(* Schneider Machine Expert - Basic project atividade2, file version 2.7.0.0 *)
(* ProjectInformations: Name=Novo projeto *)

HARDWARE
  Cpu 0: TM221CE24R
  EthernetConfiguration: NetworkName=M221, IpAllocationMode=FixedAddress, IpAddress=0.0.0.0, SubnetMask=0.0.0.0
  SerialLineConfiguration: Baud=Baud19200, Parity=ParityEven, DataBits=DataBits8, StopBits=StopBits1, PhysicalMedium=PhysicalMediumRs485, TransmissionMode=TransmissionModeModbusRtu, SlaveId=1, Addressing=SlaveAddressing
  MastTask: UsePeriodScanMode=false, PeriodScan=100
  FastTask: Period=255
  CpuBehavior: StartingMode=StartAsPreviousState, AutoSaveRamOnEeprom=true, WatchdogPeriod=250

SYMBOLS  (address, symbol, comment, settings)
  %M0       SIG_IN_SEN_A_ATU
  %M1       SIG_IN_SEN_A_DESA
  %M2       SIG_IN_SEN_B_ATU
  %M3       SIG_IN_SEN_B_DESA
  %M4       SIG_IN_SEN_C_ATU
  %M5       SIG_IN_SEN_C_DESA
  %M6       SIG_IN_SEN_D_ATU
  %M7       SIG_IN_SEN_D_DESA
  %M10      SIG_OUT_M1_LIGA
  %M11      SIG_OUT_M1_DESL
  %M12      SIG_OUT_M2_LIGA
  %M13      SIG_OUT_M2_DESL
  %M14      SIG_OUT_P1_LIGA
  %M15      SIG_OUT_P1_DESL
  %M16      SIG_OUT_AL1_LIGA
  %M17      SIG_OUT_AL1_DESL
  %M20      SIG_OUT_M1
  %M21      SIG_OUT_M2
  %M22      SIG_OUT_P1
  %M23      SIG_OUT_P2
  %M24      SIG_OUT_SEN_A
  %M25      SIG_OUT_SEN_B
  %M26      SIG_OUT_SEN_C
  %M27      SIG_OUT_SEN_D
  %M30      SIN_IN_SEL_A_ATU
  %M31      SIN_IN_SEL_A_DESA
  %M32      SIN_IN_EMERG_ATU
  %M33      SIN_IN_EMERG_DESA
  %I0.0     IN_SEN_A
  %I0.1     IN_SEN_B
  %I0.2     IN_SEN_C
  %I0.3     IN_SEN_D
  %I0.4     IN_SEL_A_ATU
  %I0.5     IN_SEL_A_DESA
  %I0.6     IN_EMERG_ATU
  %I0.7     IN_EMERG_DESA
  %Q0.0     OUT_M1
  %Q0.1     OUT_M2
  %Q0.2     OUT_P1
  %Q0.3     OUT_AL1
  %Q0.4     OUT_SEN_A
  %Q0.5     OUT_SEN_B
  %Q0.6     OUT_SEN_C
  %Q0.7     OUT_SEN_D

POU Entradas
  (* SectionNumber=1 *)

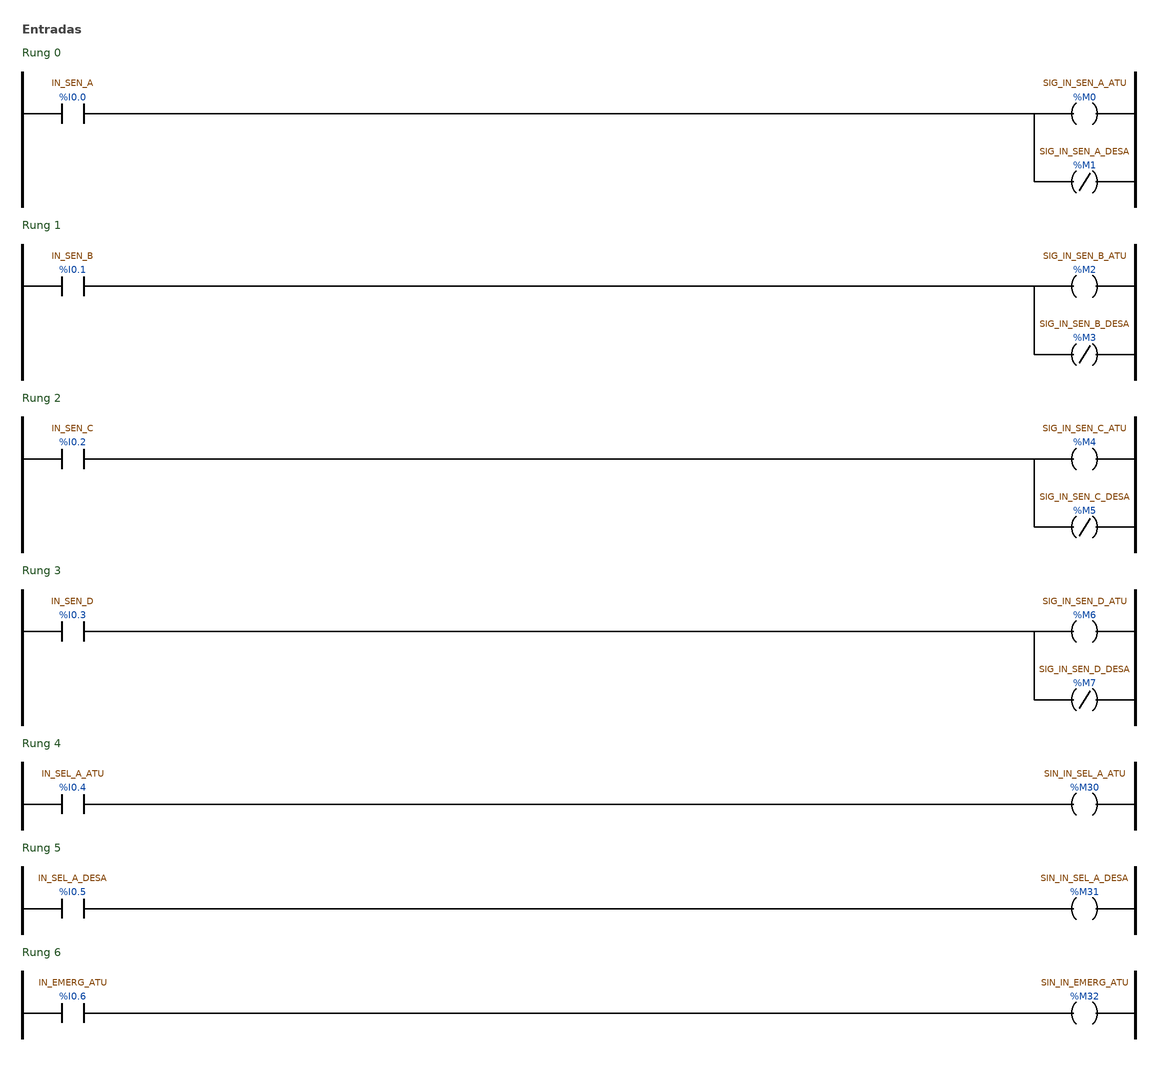

// Rung 0
  LD %I0.0                (* IN_SEN_A *)
  ST %M0                  (* SIG_IN_SEN_A_ATU *)
  STN %M1                 (* SIG_IN_SEN_A_DESA *)
  // as ST:
  //   SIG_IN_SEN_A_ATU := IN_SEN_A;
  //   SIG_IN_SEN_A_DESA := NOT IN_SEN_A;

// Rung 1
  LD %I0.1                (* IN_SEN_B *)
  ST %M2                  (* SIG_IN_SEN_B_ATU *)
  STN %M3                 (* SIG_IN_SEN_B_DESA *)
  // as ST:
  //   SIG_IN_SEN_B_ATU := IN_SEN_B;
  //   SIG_IN_SEN_B_DESA := NOT IN_SEN_B;

// Rung 2
  LD %I0.2                (* IN_SEN_C *)
  ST %M4                  (* SIG_IN_SEN_C_ATU *)
  STN %M5                 (* SIG_IN_SEN_C_DESA *)
  // as ST:
  //   SIG_IN_SEN_C_ATU := IN_SEN_C;
  //   SIG_IN_SEN_C_DESA := NOT IN_SEN_C;

// Rung 3
  LD %I0.3                (* IN_SEN_D *)
  ST %M6                  (* SIG_IN_SEN_D_ATU *)
  STN %M7                 (* SIG_IN_SEN_D_DESA *)
  // as ST:
  //   SIG_IN_SEN_D_ATU := IN_SEN_D;
  //   SIG_IN_SEN_D_DESA := NOT IN_SEN_D;

// Rung 4
  LD %I0.4                (* IN_SEL_A_ATU *)
  ST %M30                 (* SIN_IN_SEL_A_ATU *)
  // as ST:
  //   SIN_IN_SEL_A_ATU := IN_SEL_A_ATU;

// Rung 5
  LD %I0.5                (* IN_SEL_A_DESA *)
  ST %M31                 (* SIN_IN_SEL_A_DESA *)
  // as ST:
  //   SIN_IN_SEL_A_DESA := IN_SEL_A_DESA;

// Rung 6
  LD %I0.6                (* IN_EMERG_ATU *)
  ST %M32                 (* SIN_IN_EMERG_ATU *)
  // as ST:
  //   SIN_IN_EMERG_ATU := IN_EMERG_ATU;

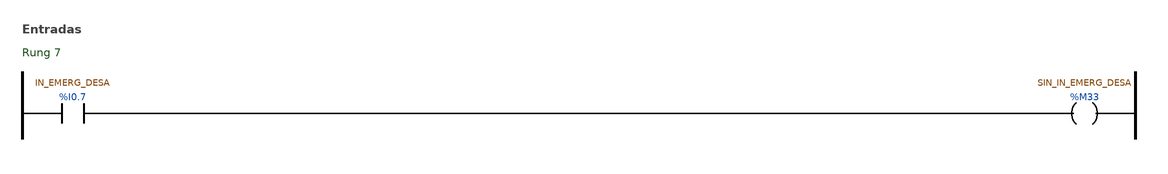

// Rung 7
  LD %I0.7                (* IN_EMERG_DESA *)
  ST %M33                 (* SIN_IN_EMERG_DESA *)
  // as ST:
  //   SIN_IN_EMERG_DESA := IN_EMERG_DESA;

POU Lógica
  (* SectionNumber=2 *)

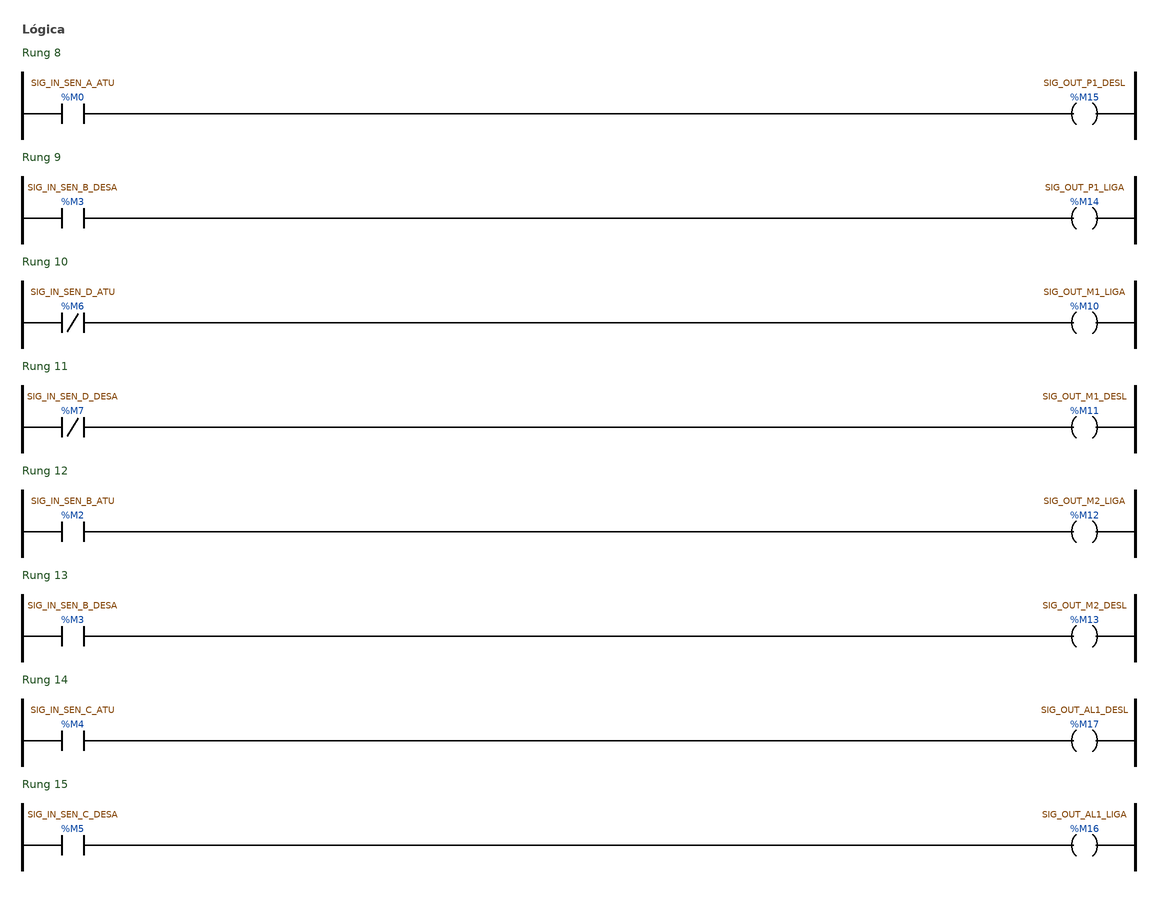

// Rung 8
  LD %M0                  (* SIG_IN_SEN_A_ATU *)
  ST %M15                 (* SIG_OUT_P1_DESL *)
  // as ST:
  //   SIG_OUT_P1_DESL := SIG_IN_SEN_A_ATU;

// Rung 9
  LD %M3                  (* SIG_IN_SEN_B_DESA *)
  ST %M14                 (* SIG_OUT_P1_LIGA *)
  // as ST:
  //   SIG_OUT_P1_LIGA := SIG_IN_SEN_B_DESA;

// Rung 10
  LDN %M6                 (* SIG_IN_SEN_D_ATU *)
  ST %M10                 (* SIG_OUT_M1_LIGA *)
  // as ST:
  //   SIG_OUT_M1_LIGA := NOT SIG_IN_SEN_D_ATU;

// Rung 11
  LDN %M7                 (* SIG_IN_SEN_D_DESA *)
  ST %M11                 (* SIG_OUT_M1_DESL *)
  // as ST:
  //   SIG_OUT_M1_DESL := NOT SIG_IN_SEN_D_DESA;

// Rung 12
  LD %M2                  (* SIG_IN_SEN_B_ATU *)
  ST %M12                 (* SIG_OUT_M2_LIGA *)
  // as ST:
  //   SIG_OUT_M2_LIGA := SIG_IN_SEN_B_ATU;

// Rung 13
  LD %M3                  (* SIG_IN_SEN_B_DESA *)
  ST %M13                 (* SIG_OUT_M2_DESL *)
  // as ST:
  //   SIG_OUT_M2_DESL := SIG_IN_SEN_B_DESA;

// Rung 14
  LD %M4                  (* SIG_IN_SEN_C_ATU *)
  ST %M17                 (* SIG_OUT_AL1_DESL *)
  // as ST:
  //   SIG_OUT_AL1_DESL := SIG_IN_SEN_C_ATU;

// Rung 15
  LD %M5                  (* SIG_IN_SEN_C_DESA *)
  ST %M16                 (* SIG_OUT_AL1_LIGA *)
  // as ST:
  //   SIG_OUT_AL1_LIGA := SIG_IN_SEN_C_DESA;

POU Lógicas Saídas
  (* SectionNumber=3 *)

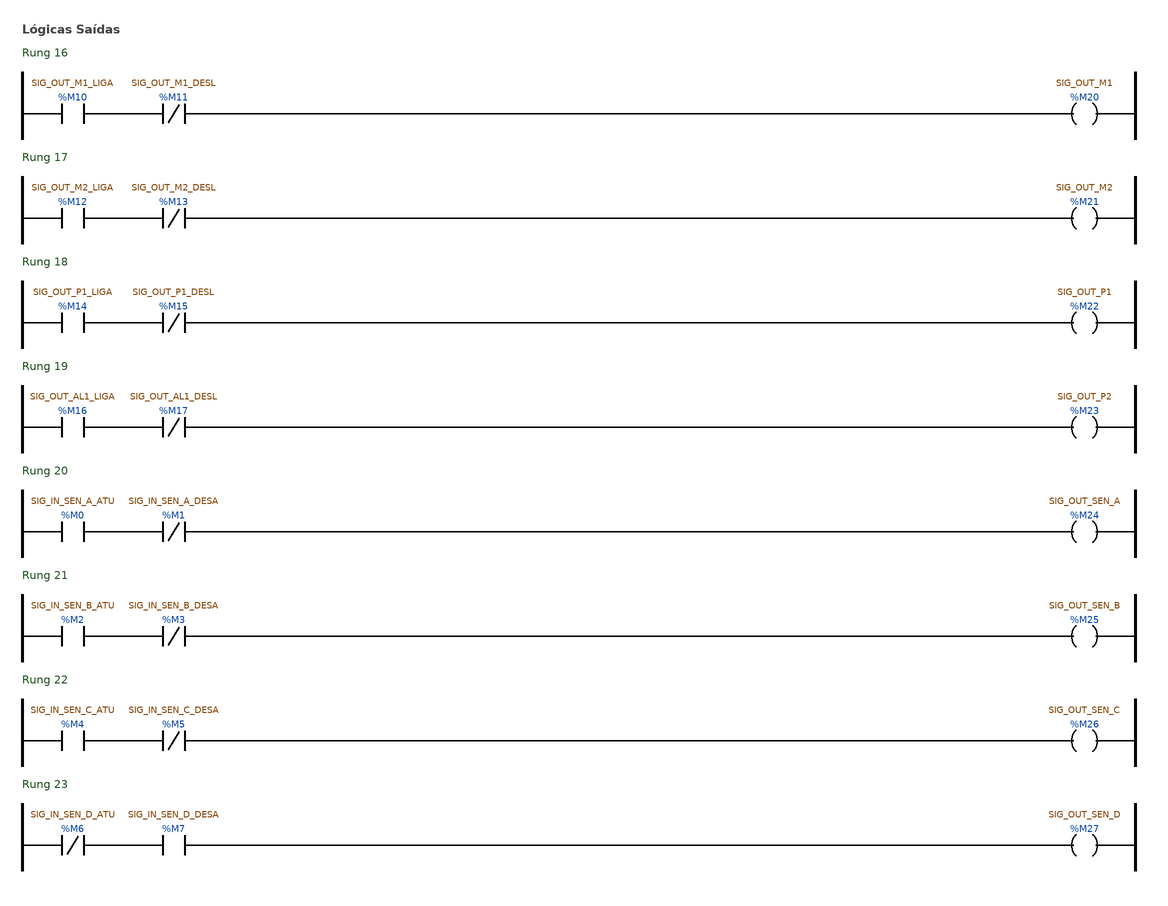

// Rung 16
  LD %M10                 (* SIG_OUT_M1_LIGA *)
  ANDN %M11               (* SIG_OUT_M1_DESL *)
  ST %M20                 (* SIG_OUT_M1 *)
  // as ST:
  //   SIG_OUT_M1 := SIG_OUT_M1_LIGA AND NOT SIG_OUT_M1_DESL;

// Rung 17
  LD %M12                 (* SIG_OUT_M2_LIGA *)
  ANDN %M13               (* SIG_OUT_M2_DESL *)
  ST %M21                 (* SIG_OUT_M2 *)
  // as ST:
  //   SIG_OUT_M2 := SIG_OUT_M2_LIGA AND NOT SIG_OUT_M2_DESL;

// Rung 18
  LD %M14                 (* SIG_OUT_P1_LIGA *)
  ANDN %M15               (* SIG_OUT_P1_DESL *)
  ST %M22                 (* SIG_OUT_P1 *)
  // as ST:
  //   SIG_OUT_P1 := SIG_OUT_P1_LIGA AND NOT SIG_OUT_P1_DESL;

// Rung 19
  LD %M16                 (* SIG_OUT_AL1_LIGA *)
  ANDN %M17               (* SIG_OUT_AL1_DESL *)
  ST %M23                 (* SIG_OUT_P2 *)
  // as ST:
  //   SIG_OUT_P2 := SIG_OUT_AL1_LIGA AND NOT SIG_OUT_AL1_DESL;

// Rung 20
  LD %M0                  (* SIG_IN_SEN_A_ATU *)
  ANDN %M1                (* SIG_IN_SEN_A_DESA *)
  ST %M24                 (* SIG_OUT_SEN_A *)
  // as ST:
  //   SIG_OUT_SEN_A := SIG_IN_SEN_A_ATU AND NOT SIG_IN_SEN_A_DESA;

// Rung 21
  LD %M2                  (* SIG_IN_SEN_B_ATU *)
  ANDN %M3                (* SIG_IN_SEN_B_DESA *)
  ST %M25                 (* SIG_OUT_SEN_B *)
  // as ST:
  //   SIG_OUT_SEN_B := SIG_IN_SEN_B_ATU AND NOT SIG_IN_SEN_B_DESA;

// Rung 22
  LD %M4                  (* SIG_IN_SEN_C_ATU *)
  ANDN %M5                (* SIG_IN_SEN_C_DESA *)
  ST %M26                 (* SIG_OUT_SEN_C *)
  // as ST:
  //   SIG_OUT_SEN_C := SIG_IN_SEN_C_ATU AND NOT SIG_IN_SEN_C_DESA;

// Rung 23
  LDN %M6                 (* SIG_IN_SEN_D_ATU *)
  AND %M7                 (* SIG_IN_SEN_D_DESA *)
  ST %M27                 (* SIG_OUT_SEN_D *)
  // as ST:
  //   SIG_OUT_SEN_D := NOT SIG_IN_SEN_D_ATU AND SIG_IN_SEN_D_DESA;

POU Saídas
  (* SectionNumber=4 *)

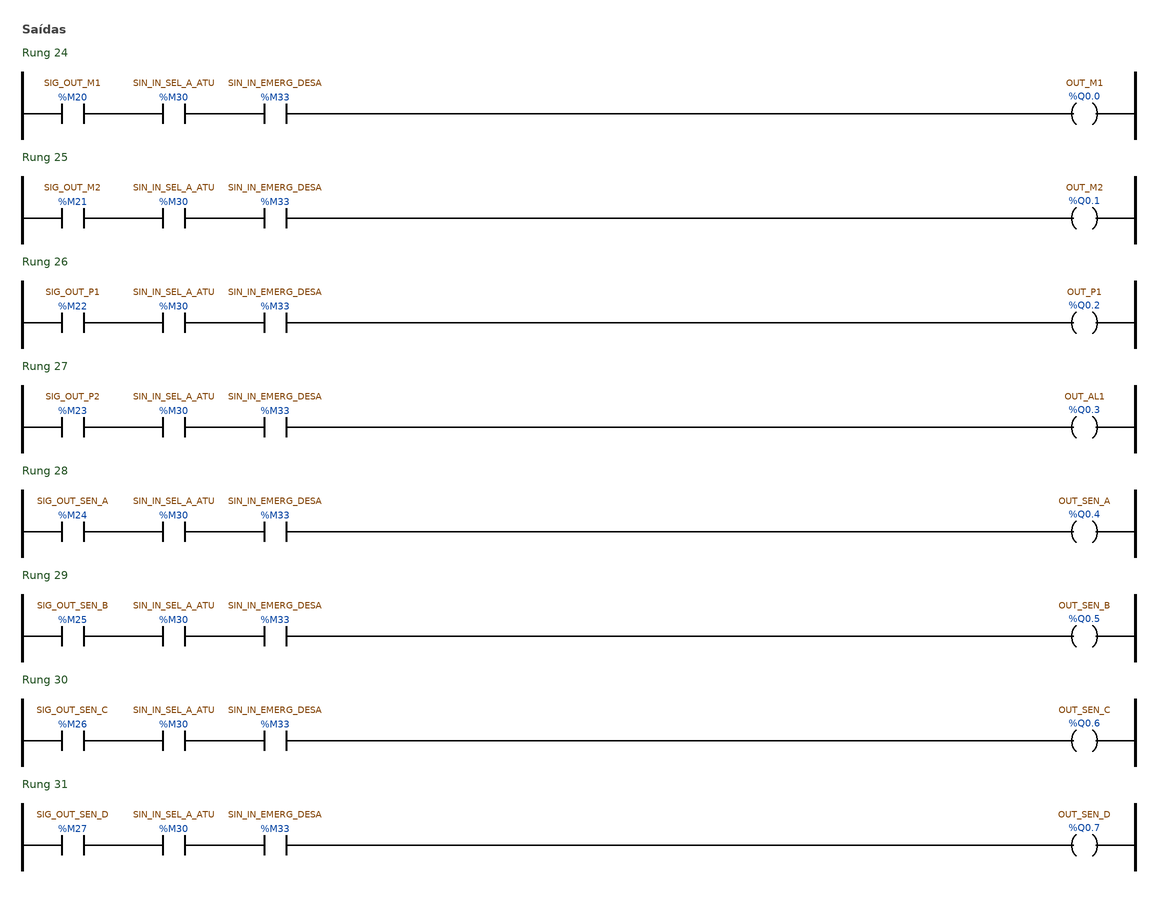

// Rung 24
  LD %M20                 (* SIG_OUT_M1 *)
  AND %M30                (* SIN_IN_SEL_A_ATU *)
  AND %M33                (* SIN_IN_EMERG_DESA *)
  ST %Q0.0                (* OUT_M1 *)
  // as ST:
  //   OUT_M1 := SIG_OUT_M1 AND SIN_IN_SEL_A_ATU AND SIN_IN_EMERG_DESA;

// Rung 25
  LD %M21                 (* SIG_OUT_M2 *)
  AND %M30                (* SIN_IN_SEL_A_ATU *)
  AND %M33                (* SIN_IN_EMERG_DESA *)
  ST %Q0.1                (* OUT_M2 *)
  // as ST:
  //   OUT_M2 := SIG_OUT_M2 AND SIN_IN_SEL_A_ATU AND SIN_IN_EMERG_DESA;

// Rung 26
  LD %M22                 (* SIG_OUT_P1 *)
  AND %M30                (* SIN_IN_SEL_A_ATU *)
  AND %M33                (* SIN_IN_EMERG_DESA *)
  ST %Q0.2                (* OUT_P1 *)
  // as ST:
  //   OUT_P1 := SIG_OUT_P1 AND SIN_IN_SEL_A_ATU AND SIN_IN_EMERG_DESA;

// Rung 27
  LD %M23                 (* SIG_OUT_P2 *)
  AND %M30                (* SIN_IN_SEL_A_ATU *)
  AND %M33                (* SIN_IN_EMERG_DESA *)
  ST %Q0.3                (* OUT_AL1 *)
  // as ST:
  //   OUT_AL1 := SIG_OUT_P2 AND SIN_IN_SEL_A_ATU AND SIN_IN_EMERG_DESA;

// Rung 28
  LD %M24                 (* SIG_OUT_SEN_A *)
  AND %M30                (* SIN_IN_SEL_A_ATU *)
  AND %M33                (* SIN_IN_EMERG_DESA *)
  ST %Q0.4                (* OUT_SEN_A *)
  // as ST:
  //   OUT_SEN_A := SIG_OUT_SEN_A AND SIN_IN_SEL_A_ATU AND SIN_IN_EMERG_DESA;

// Rung 29
  LD %M25                 (* SIG_OUT_SEN_B *)
  AND %M30                (* SIN_IN_SEL_A_ATU *)
  AND %M33                (* SIN_IN_EMERG_DESA *)
  ST %Q0.5                (* OUT_SEN_B *)
  // as ST:
  //   OUT_SEN_B := SIG_OUT_SEN_B AND SIN_IN_SEL_A_ATU AND SIN_IN_EMERG_DESA;

// Rung 30
  LD %M26                 (* SIG_OUT_SEN_C *)
  AND %M30                (* SIN_IN_SEL_A_ATU *)
  AND %M33                (* SIN_IN_EMERG_DESA *)
  ST %Q0.6                (* OUT_SEN_C *)
  // as ST:
  //   OUT_SEN_C := SIG_OUT_SEN_C AND SIN_IN_SEL_A_ATU AND SIN_IN_EMERG_DESA;

// Rung 31
  LD %M27                 (* SIG_OUT_SEN_D *)
  AND %M30                (* SIN_IN_SEL_A_ATU *)
  AND %M33                (* SIN_IN_EMERG_DESA *)
  ST %Q0.7                (* OUT_SEN_D *)
  // as ST:
  //   OUT_SEN_D := SIG_OUT_SEN_D AND SIN_IN_SEL_A_ATU AND SIN_IN_EMERG_DESA;
